// TIA Portal project "Temporizadores" (V15)

(* hardware
DEVICE "S7-1200 station_1"  S7-1200 Station
   slot 0: "Rack_0"  S7-1200 Rack  Rack  V1.0
   slot 1: "PLC_1"  CPU 1214C DC/DC/DC  6ES7 214-1AG40-0XB0  V4.2
*)

// ===== PLC "PLC_1"  CPU 1214C DC/DC/DC =====

VAR_GLOBAL   // PLC tag table "Tabla de variables estándar"
   "System_Byte" AT %MB0 : Byte;
   "FirstScan" AT %M0.0 : Bool;
   "DiagStatusUpdate" AT %M0.1 : Bool;
   "AlwaysTRUE" AT %M0.2 : Bool;
   "AlwaysFALSE" AT %M0.3 : Bool;
   "Clock_Byte" AT %MB0 : Byte;
   "Clock_10Hz" AT %M0.0 : Bool;
   "Clock_5Hz" AT %M0.1 : Bool;
   "Clock_2.5Hz" AT %M0.2 : Bool;
   "Clock_2Hz" AT %M0.3 : Bool;
   "Clock_1.25Hz" AT %M0.4 : Bool;
   "Clock_1Hz" AT %M0.5 : Bool;
   "Clock_0.625Hz" AT %M0.6 : Bool;
   "Clock_0.5Hz" AT %M0.7 : Bool;
   "Marcha" AT %I0.0 : Bool;
   "Paro" AT %I0.1 : Bool;
   "Termoestato" AT %I0.2 : Bool;
   "C_Bomba" AT %Q0.0 : Bool;
   "Sisema_Activo" AT %M10.0 : Bool;
   "OL" AT %I0.3 : Bool;
   "Alarma_Bomba" AT %Q0.1 : Bool;
   "Start1" AT %I0.4 : Bool;
   "Motor1" AT %Q0.2 : Bool;
   "Tag_1" AT %I0.5 : Bool;
   "Motor 2" AT %Q0.3 : Bool;
   "Tag_2" AT %I0.6 : Bool;
   "Tiempo Reposo" AT %MD20 : Time;
   "Motor 3" AT %Q0.4 : Bool;
   "Tag_3" AT %I0.7 : Bool;
   "Motor 4" AT %Q0.5 : Bool;
   "Tag_4" AT %I1.0 : Bool;
END_VAR

// folder: System blocks/Program resources

DATA_BLOCK "T_Trabajo"   // DB1
{ S7_Optimized_Access := 'TRUE' }
AUTHOR : Simatic
FAMILY : IEC
NAME : IEC_TMR
VERSION : 1.0
// stored: InstanceOfName IEC_TIMER
"IEC_TIMER"
BEGIN
END_DATA_BLOCK

DATA_BLOCK "Impulso"   // DB2
{ S7_Optimized_Access := 'TRUE' }
AUTHOR : Simatic
FAMILY : IEC
NAME : IEC_TMR
VERSION : 1.0
// stored: InstanceOfName IEC_TIMER
"IEC_TIMER"
BEGIN
END_DATA_BLOCK

DATA_BLOCK "Reposo"   // DB3
{ S7_Optimized_Access := 'TRUE' }
AUTHOR : Simatic
FAMILY : IEC
NAME : IEC_TMR
VERSION : 1.0
// stored: InstanceOfName IEC_TIMER
"IEC_TIMER"
BEGIN
END_DATA_BLOCK

DATA_BLOCK "Horometro"   // DB4
{ S7_Optimized_Access := 'TRUE' }
AUTHOR : Simatic
FAMILY : IEC
NAME : IEC_TMR
VERSION : 1.0
// stored: InstanceOfName IEC_TIMER
"IEC_TIMER"
BEGIN
END_DATA_BLOCK

// folder: (top level)

FUNCTION "Control_Enfriamiento" : Void   // FC1, LAD
{ S7_Optimized_Access := 'TRUE' }
VERSION : 0.1
BEGIN

REGION Network 1
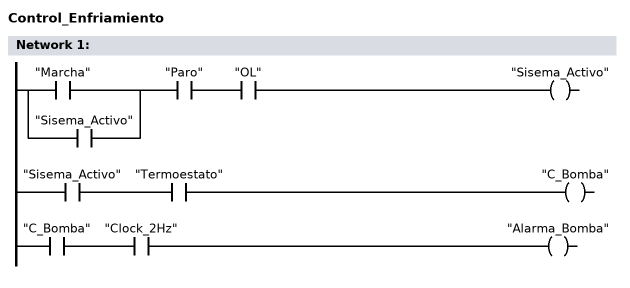
   RUNG wire#powerrail
      Contact( "Marcha" )
      wire#w1
      Contact( "Paro" )
      Contact( "OL" )
      Coil( "Sisema_Activo" )
   END_RUNG
   RUNG wire#powerrail
      Contact( "Sisema_Activo" )
   END_RUNG wire#w1
   RUNG wire#powerrail
      Contact( "Sisema_Activo" )
      Contact( "Termoestato" )
      Coil( "C_Bomba" )
   END_RUNG
   RUNG wire#powerrail
      Contact( "C_Bomba" )
      Contact( "Clock_2Hz" )
      Coil( "Alarma_Bomba" )
   END_RUNG
   // the same network as SCL:
   "Sisema_Activo" := ("Marcha" OR "Sisema_Activo") AND "Paro" AND "OL";
   "C_Bomba" := "Sisema_Activo" AND "Termoestato";
   "Alarma_Bomba" := "C_Bomba" AND "Clock_2Hz";
END_REGION
END_FUNCTION

FUNCTION "Temporizadores" : Void   // FC2, LAD
{ S7_Optimized_Access := 'TRUE' }
VERSION : 0.1
BEGIN

REGION Network 1
   // Temporizador al rabajo
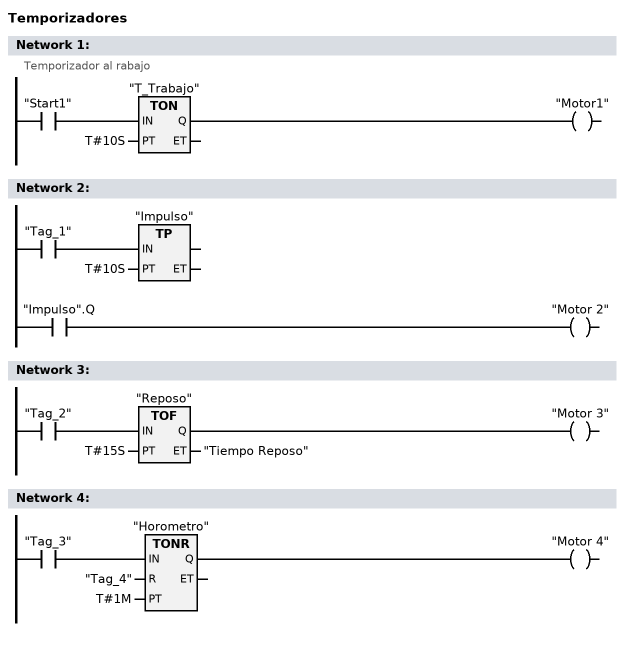
   "T_Trabajo".TON(IN := "Start1", PT := T#10S);
   "Motor1" := "T_Trabajo".Q;
END_REGION

REGION Network 2
   "Impulso".TP(IN := "Tag_1", PT := T#10S);
   "Motor 2" := "Impulso".Q;
END_REGION

REGION Network 3
   "Reposo".TOF(IN := "Tag_2", PT := T#15S, ET => "Tiempo Reposo");
   "Motor 3" := "Reposo".Q;
END_REGION

REGION Network 4
   "Horometro".TONR(IN := "Tag_3", R := "Tag_4", PT := T#1M);
   "Motor 4" := "Horometro".Q;
END_REGION
END_FUNCTION

ORGANIZATION_BLOCK "Main"   // OB1, LAD, ProgramCycle
TITLE = "Main Program Sweep (Cycle)"
{ S7_Optimized_Access := 'TRUE' }
VERSION : 0.1
   VAR_INPUT
      Initial_Call : Bool;   // Initial call of this OB
      Remanence : Bool;   // =True, if remanent data are available
   END_VAR
BEGIN

REGION Network 1
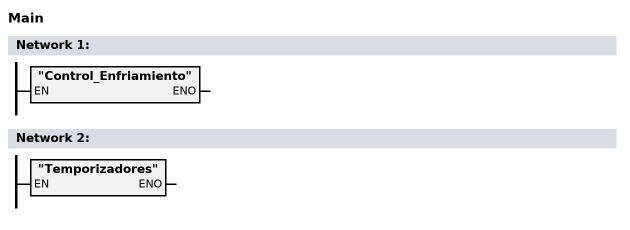
   RUNG wire#powerrail
      "Control_Enfriamiento"()
   END_RUNG
   // the same network as SCL:
   "Control_Enfriamiento"();
END_REGION

REGION Network 2
   RUNG wire#powerrail
      "Temporizadores"()
   END_RUNG
   // the same network as SCL:
   "Temporizadores"();
END_REGION
END_ORGANIZATION_BLOCK